// TIA Portal V16 export
// export: Created 2023-03-29T11:03:35.6788422Z, ExportSetting WithDefaults, DisplayName Totally Integrated Automation Portal, DisplayVersion V16 Update 6, DisplayName TIA Portal Version Control Interface, DisplayVersion V16 Update 2, DisplayName TIA Portal Openness, DisplayVersion V16 Update 6, DisplayName STEP 7 Professional, DisplayVersion V16 Update 6, DisplayName STEP 7 Safety, DisplayVersion V16, DisplayName WinCC Advanced, DisplayVersion V16 Update 6
DATA_BLOCK "V_ErrorOB"   // DB108
{ S7_Optimized_Access := 'TRUE' }
VERSION : 0.1
// stored: AutoNumber false, DBAccessibleFromOPCUA true, IsOnlyStoredInLoadMemory false, IsRetainMemResEnabled false, IsWriteProtectedInAS false, MemoryReserve 0
   VAR
      StartUp { S7_SetPoint := 'True'} : "stt_ERR_StartUpOB";   // //Error read in OB100
      OB80 : Bool;   // //Executed OB80 Time error interrupt
      ResetErrorOB : Bool;   // //Variable connected with button in web site
   END_VAR
BEGIN
END_DATA_BLOCK
